INTERFACE I_AxisStatus EXTENDS __SYSTEM.IQueryInterface

METHOD getCurrentPosition : LREAL
VAR_INPUT
END_VAR
END_METHOD

METHOD isAtPosition : BOOL
VAR_INPUT
	position : MC_LREAL;
END_VAR
END_METHOD

METHOD isInVelocity : BOOL
VAR_INPUT
	Velocity : MC_LREAL;
END_VAR
END_METHOD

METHOD isStationary : BOOL
VAR_INPUT
END_VAR
END_METHOD

END_INTERFACE

(* stored: Version 1.1.0.1
   Itf I_AxisStatus: Id {6057db56-1d8d-4c90-8f15-4379a266ab62}
   Method getCurrentPosition: Id {4fa41b0c-b611-436e-9bd7-2a6e55e87dc6}
   Method isAtPosition: Id {b1b2fe74-f8e0-4241-b0e9-3e1b63b14a12}
   Method isInVelocity: Id {3b580483-8069-42c2-961f-3563b2202ac4}
   Method isStationary: Id {58e66eb5-9088-44a9-a122-982f73f5789e} *)
